FUNCTION_BLOCK MECH_VIEWER (* Linear Mechanism View with Local Data Publish/Subscribe *)
  (* Standard: 61499-1; Classification: View *)
  (* Version 0.4, 2010-11-13, JHC, Holobloc Inc, Removed duplicated connections (?). Added hmi import for VDIR. *)
  (* Version 0.3, 2010-11-07, JHC, Holobloc Inc, Changed DIR type to VDIR. *)
  (* Version 0.2, 2002-05-02, JHC, Rockwell Automation, Changed to optimized PUBL/SUBL, standardized IDs. *)
  (* Version 0.1, 2002-04-21, JHC, Rockwell Automation, Changed PUBL/SUBL to PUBLISH/SUBSCRIBE. *)
  (* Version 0.0, 2002-04-14, JHC, Rockwell Automation *)
  (* Compiler header: package fb.rt.mva; import fb.rt.net.*; import fb.rt.hmi.*; *)
  (* Compiler classdef: public class MECH_VIEWL extends FBMVCD *)
  (* Compiler Java IBM VisualAge 3.0 *)
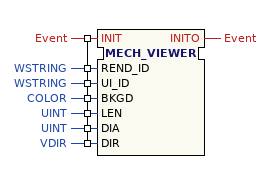
  EVENT_INPUT
    INIT WITH REND_ID, UI_ID, BKGD, LEN, DIA, DIR; (* Initialize *)
  END_EVENT
  EVENT_OUTPUT
    INITO; (* Initialized *)
  END_EVENT
  VAR_INPUT
    REND_ID : WSTRING; (* Rendering Data Channel from Model *)
    UI_ID : WSTRING; (* User Input Channel to Model *)
    BKGD : COLOR := blue; (* Background Color *)
    LEN : UINT; (* Length in Diameters *)
    DIA : UINT; (* Diameter *)
    DIR : VDIR; (* Orientation *)
  END_VAR
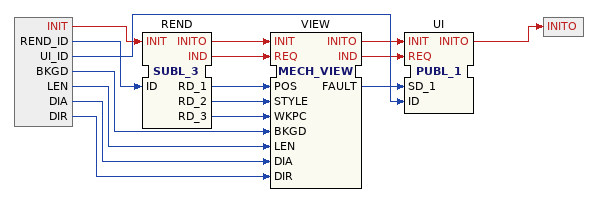
  FBS
    REND : SUBL_3;
    VIEW : MECH_VIEW;
    UI : PUBL_1;
  END_FBS
  EVENT_CONNECTIONS
    INIT TO REND.INIT;
    REND.INITO TO VIEW.INIT;
    VIEW.INITO TO UI.INIT;
    UI.INITO TO INITO;
    REND.IND TO VIEW.REQ;
    VIEW.IND TO UI.REQ;
  END_CONNECTIONS
  DATA_CONNECTIONS
    REND.RD_1 TO VIEW.POS;
    REND.RD_2 TO VIEW.STYLE;
    REND.RD_3 TO VIEW.WKPC;
    VIEW.FAULT TO UI.SD_1;
    REND_ID TO REND.ID;
    UI_ID TO UI.ID;
    BKGD TO VIEW.BKGD;
    LEN TO VIEW.LEN;
    DIA TO VIEW.DIA;
    DIR TO VIEW.DIR;
  END_CONNECTIONS
END_FUNCTION_BLOCK
